{attribute 'GeneratedUsingTerminal: EL3174-0002-0017'}
{attribute addProperty BoxType "EL3174-0002-0017"}
{attribute addProperty Id "StatusAT %I*Status_B07533568ValueAT %I*INT2"}
{attribute addProperty CRC "2833212643"}
{attribute addProperty Size "10"}
TYPE AI_Standard_Channel_A8DF64E3 EXTENDS TcoIo.InputBase_8311D824 :
STRUCT
	{attribute addProperty Name "Status"}
	Status AT %I* : Status_B0753356;
	{attribute addProperty Name "Value"}
	Value AT %I* : INT;
END_STRUCT
END_TYPE

(* stored: Version 1.2.0.0, ProductVersion 3.1.4024.11
   DUT AI_Standard_Channel_A8DF64E3: Id {de54ded0-fbac-0233-1686-129baf37c638} *)
